FUNCTION_BLOCK FB_Object_List_Testing
VAR_INPUT
	Start			: BOOL;	
	Complete_test	: BOOL := FALSE;	
	RPDO_Nr			: BYTE := 0;
	TPDO_Nr			: BYTE := 0;
END_VAR
VAR_IN_OUT
	Object_List		: ARRAY [*] OF ST_CAN_Object;
END_VAR
VAR_OUTPUT
	Finished		: BOOL := FALSE;
	Error			: BOOL := FALSE;
END_VAR
VAR
	State			: INT := 0;	
	Index 			: BYTE := 0;
	i 				: DINT := 0;
	
	Object_Testing	: FB_Object_Testing;

	SubIndex_Count	: BYTE := 0;
END_VAR

IF Start AND State = 255 THEN 
	Finished 	:= FALSE;
	Error 		:= FALSE;
	State 		:= 0;
END_IF


CASE State OF	
	0:	// Start check objects	
	IF Start THEN
		Object_Testing(CAN_Object:=Object_List[0], Start:=TRUE, Complete_test:=TRUE, RPDO_Nr:=3, TPDO_Nr:=3);
		Index := 0;
		
		State := State + 1;
	END_IF
	
	
	1:	// Running, wait for finish and start next object
	Object_Testing(CAN_Object:=Object_List[Index], Start:=FALSE);
	
	IF Object_Testing.Finished THEN
		
		CASE Object_List[Index].SubElements OF
			E_SubElement_types.With_fix_subelements:	// Object with fix subelements
				IF (Object_List[Index].Readable) AND ((Object_List[Index].Read_Value > 0) OR (Object_List[Index +1].Mandatory > 0)) THEN
					Index := Index + 1;
				ELSE
					Index := Index + 1 + DWORD_TO_BYTE(Object_List[Index].Default_Value);
				END_IF	 						
				
								
			E_SubElement_types.Fix_subelement:	// Next object
				Index := Index + 1;		
					
	
			E_SubElement_types.With_list:		// Object with a variable count of subelements	
				IF Object_List[Index].Readable AND Object_List[Index].Read_Value > 0 THEN
					Index := Index + 1;						
					Object_List[Index].Subindex := 1;
				ELSE
					Index := Index + 2;
				END_IF


			E_SubElement_types.List_element:	// Next variable subobject or next object
				IF Object_List[Index - 1].Read_Value > Object_List[Index].Subindex  THEN
					Object_List[Index].Subindex := Object_List[Index].Subindex + 1;
				ELSE
					Index := Index + 1;	
				END_IF
			
			
			E_SubElement_types.No:	// Standalone object -> next object
				Index := Index + 1;
					
	
			ELSE					// Unknown Type -> next object
				Index := Index + 1;
						
		END_CASE
		
		// Test next Object
		IF Index <= UPPER_BOUND(Object_List,1) THEN 
			Object_Testing(CAN_Object:=Object_List[Index], Start:=TRUE, Complete_test:=TRUE, RPDO_Nr:=3, TPDO_Nr:=3);	
		ELSE			
			State := 254;
		END_IF		
	END_IF	
	
	
	// ************ Finished ************			
	254: // Check error 
		Error := FALSE;
		FOR i := 0 TO UPPER_BOUND(Object_List,1) DO
			Error := Error OR Object_List[i].Error;			
		END_FOR;
		Finished := TRUE;	
		State := 255;
		
	255: // Tests finished
		Finished := TRUE;
	

	ELSE		
		State := 254;
		
END_CASE

END_FUNCTION_BLOCK

(* stored: Version 1.1.0.1, ProductVersion 3.1.4024.11
   POU FB_Object_List_Testing: Id {ca66eaee-c343-4caa-95ba-6a980cd0d9b1}, SpecialFunc None *)
